TYPE ST_LightTowerAction :
STRUCT
	GREEN			: BOOL;
	GREEN_FLASHING	: BOOL;
	
	RED				: BOOL;
	RED_FLASHING	: BOOL;
	
	YELLOW			: BOOL;
	YELLOW_FLASHING	: BOOL;
	
	BLUE			: BOOL;
	BLUE_FLASHING	: BOOL;
	
	WHITE			: BOOL;
	WHITE_FLASHING	: BOOL;
	
	BEEPING			: BOOL;
	BEEPING_FLASHING: BOOL;
END_STRUCT
END_TYPE

(* stored: Version 1.1.0.1, ProductVersion 3.1.4024.12
   DUT ST_LightTowerAction: Id {d086dee9-590d-4737-ab6f-ce742ffc4750} *)
